PROGRAM PRG_GEM1
VAR
	{attribute 'pytmc' :=' pv: EM1L0:GEM:CNTRL:RESET;
     field: ZNAM FALSE; 
	 field: ONAM TRUE; 
	 io: io;
	'}
	bReset : BOOL; 
	{attribute 'pytmc' :=' pv: EM1L0:GEM:CNTRL:ERROR;
     field: ZNAM FALSE; 
	 field: ONAM TRUE; 
	 io: io;
	'}
	bError : BOOL; 
	{attribute 'pytmc' :=' pv: EM1L0:GEM:CNTRL:Kp1 '}
	fKp1 : REAL:= 0.5; 
	{attribute 'pytmc' :=' pv: EM1L0:GEM:CNTRL:Tn1 '}
	fTn1 : REAL:= 0.5; 
	{attribute 'pytmc' :=' pv: EM1L0:GEM:CNTRL:Kp2 '}
	fKp2 : REAL:= 0.01; 
	{attribute 'pytmc' :=' pv: EM1L0:GEM:CNTRL:Tn2 '}
	fTn2 : REAL:= 0.5; 
	arrTable_GEM1	: ARRAY[1..31,1..2] OF FLOAT;
	fManValue											: FLOAT;
	bExtrapolate										: BOOL;
	eMode							: E_CTRL_MODE;
	stCTRL_PID_PARAMS		: ST_CTRL_PID_PARAMS;
	bSync							: BOOL;
	bHold							: BOOL;
	eErrorId						: E_CTRL_ERRORCODES;
	bARWactive					: BOOL;
	(* controller *)
	fbCTRL_PID					: FB_CTRL_PID;
	bInit							: BOOL	:= TRUE;
	fbCTRL_LIN_INTERPOLATION					: FB_CTRL_LIN_INTERPOLATION;
	//stCTRL_LIN_INTERPOLATION_PARAMS		: ST_CTRL_LIN_INTERPOLATION_PARAMS;
	stCTRL_LIN_INTERPOLATION_PARAMS_GEM	: ST_CTRL_LIN_INTERPOLATION_PARAMS;
	fbCTRL_DEADBAND						: FB_CTRL_DEADBAND;
	stCTRL_DEADBAND_PARAMS			: ST_CTRL_DEADBAND_PARAMS;
		//timer to switch the pid from manual to active 5seconds??? 10 seconds???
	pid_on :TON;
	wait : time := T#10S;
FTrig: F_TRIG;	
	
	
END_VAR


(*Devices*)
(* GEM 1*)
(*Gauges*)
GEM1_GCM_41(i_rFULL_SCALE := 10.0 (*Torr*));
GEM1_GCM_42(i_rFULL_SCALE := 0.05 (*Torr*));
(*Assign reading to psuedo gauge*)
IF (GEM1_GCM_42.PG.rPRESS >0.04) THEN GEM1_GCM_40 := GEM1_GCM_42.PG;
	ELSE
	GEM1_GCM_40 := GEM1_GCM_41.PG;	
END_IF
(* N2 Cut Off Valves *)
GEM1_VVC_40(i_xExtILK_OK:= GEM1_Aperture_Closed AND GEM1_Turbo_Valves_Open AND GEM1_Turbo_Running); 

(*Flow Control Valves*)
GEM1_VCN_40 (i_xExtIlkOK := (GEM1_Aperture_Closed AND GEM1_Turbo_Valves_Open AND GEM1_Turbo_Running),// AND  GEM1_VVC_40.M_IsOpen()),
			 i_ReqPos:= fbCTRL_LIN_INTERPOLATION.fOut + fbCTRL_PID.fOut);
//GEM1_VPC_42 (i_xExtIlkOK := TRUE, i_rReqPos:= );



(*Iniitialization*)
IF bInit
THEN
	
	
	(* init array with the interpolation points  *)
	(* 	fIn					 |		fOut		*)
	arrTable_GEM1[1,1] := 0;		arrTable_GEM1[1,2] := 0;
	arrTable_GEM1[2,1] := 0.00178;		arrTable_GEM1[2,2] := 30;
	arrTable_GEM1[3,1] := 0.0025;		arrTable_GEM1[3,2] := 32;
	arrTable_GEM1[4,1] :=  0.003;	    arrTable_GEM1[4,2] := 34;
	arrTable_GEM1[5,1] :=  0.005884;	    arrTable_GEM1[5,2] := 35;
	arrTable_GEM1[6,1] := 0.0045;		arrTable_GEM1[6,2] := 42;
	arrTable_GEM1[7,1] := 0.09;		arrTable_GEM1[7,2] := 45;
	arrTable_GEM1[8,1] := 0.1;	    arrTable_GEM1[8,2] := 46;
	arrTable_GEM1[9,1] := 0.152;	    arrTable_GEM1[9,2] := 47;
	arrTable_GEM1[10,1] := 0.199;		arrTable_GEM1[10,2] := 50;
	arrTable_GEM1[11,1] := 0.24;		arrTable_GEM1[11,2] := 52;
	arrTable_GEM1[12,1] := 0.29;		arrTable_GEM1[12,2] := 54;
	arrTable_GEM1[13,1] := 0.3;		arrTable_GEM1[13,2] := 56;
	arrTable_GEM1[14,1] := 0.39;		arrTable_GEM1[14,2] := 56.5;
	arrTable_GEM1[15,1] := 0.6;		arrTable_GEM1[15,2] := 58;
	arrTable_GEM1[16,1] := 0.6929;		arrTable_GEM1[16,2] := 60;
	arrTable_GEM1[17,1] := 0.7322;		arrTable_GEM1[17,2] := 62;
	arrTable_GEM1[18,1] := 0.7928;	    arrTable_GEM1[18,2] := 64;
	arrTable_GEM1[19,1] := 0.85;;	    arrTable_GEM1[19,2] :=66;
	arrTable_GEM1[20,1] := 0.91;		arrTable_GEM1[20,2] := 68;
	arrTable_GEM1[21,1] := 1;		arrTable_GEM1[21,2] := 69;
	arrTable_GEM1[22,1] :=  1.0448;	    arrTable_GEM1[22,2] := 70;
	arrTable_GEM1[23,1] :=  1.31919;	    arrTable_GEM1[23,2] := 72;
	arrTable_GEM1[24,1] :=1.324;		arrTable_GEM1[24,2] := 73.04;
	arrTable_GEM1[25,1] :=1.71941;		arrTable_GEM1[25,2] := 73.64;
	arrTable_GEM1[26,1] := 1.81941;		arrTable_GEM1[26,2] := 74.45;
	arrTable_GEM1[27,1] :=  1.963194;		arrTable_GEM1[27,2] :=74.46;
	arrTable_GEM1[28,1] := 1.99999;	arrTable_GEM1[28,2] := 75;
	arrTable_GEM1[29,1] :=  2;		arrTable_GEM1[29,2] :=75.5;
	arrTable_GEM1[30,1] := 2.1;	arrTable_GEM1[30,2] := 75.505;
	arrTable_GEM1[31,1] := 2.2;	arrTable_GEM1[31,2] := 75.55;
	
	(* init parameter struct *)
	stCTRL_LIN_INTERPOLATION_PARAMS_GEM.tCtrlCycleTime					:= T#10ms;
	stCTRL_LIN_INTERPOLATION_PARAMS_GEM.tTaskCycleTime					:= T#10ms;
	stCTRL_LIN_INTERPOLATION_PARAMS_GEM.nDataTable_NumberOfRows		:= INT_TO_UINT(31);	


	(* init parameter struct *)
	stCTRL_PID_PARAMS.tCtrlCycleTime		:= T#10ms;
	stCTRL_PID_PARAMS.tTaskCycleTime		:= T#10ms;
	stCTRL_PID_PARAMS.fKp					:= fKp1;			(* proportional gain Kp				*)
	stCTRL_PID_PARAMS.tTn					:= T#1s;		(*  Tn									*)
	stCTRL_PID_PARAMS.tTv					:= T#200ms;	(*  Tv									*)
	stCTRL_PID_PARAMS.tTd					:= T#100ms;	(*  Td									*)
	stCTRL_PID_PARAMS.fOutMaxLimit			:=  78;			(* maximum output limit				*)
	stCTRL_PID_PARAMS.fOutMinLimit			:=  -100;			(* minimum output limit				*)

	(* set the mode to ACTIVE --> normal operation *)
	eMode							:= eCTRL_MODE_PASSIVE    ;					
	(* reset the init flag *)
	bInit							:= FALSE;
END_IF
(* set the addresses *)
stCTRL_LIN_INTERPOLATION_PARAMS_GEM.pDataTable_ADR			:= ADR(arrTable_GEM1);
stCTRL_LIN_INTERPOLATION_PARAMS_GEM.nDataTable_SIZEOF		:= SIZEOF(arrTable_GEM1);



if (GEM1_GO) THEN
	IF (bReset) THEN
		(* set the mode to RESET*)
		eMode							:= eCTRL_MODE_RESET   ;
		GEM1_VCN_40.M_ValveControl(CloseValve);
		//bReset := False;
	ELSE(* set the mode to ACTIVE --> normal operation *)
		eMode							:= eCTRL_MODE_ACTIVE   ;
		GEM1_VCN_40.M_ValveControl(PressureControl);
	END_IF
END_IF

If(FTrig.Q)THEN
		eMode							:= eCTRL_MODE_PASSIVE;
		GEM1_VCN_40.M_ValveControl(CloseValve);
		fGEM1SetpointValue :=0;
END_IF


fbCTRL_LIN_INTERPOLATION(
	fIn:= fGEM1SetpointValue , 
	fManValue:= fManValue, 
	bExtrapolate:= bExtrapolate, 
	eMode:= eMode, 
	fOut=> , 
	bInIsGreaterThanMaxElement=> , 
	bInIsLessThanMinElement=> , 
	eState=> , 
	eErrorId=> , 
	bError=> , 
	stParams:= stCTRL_LIN_INTERPOLATION_PARAMS_GEM );
	
(* Gauge selection *)
IF (fGEM1SetpointValue >0.04) THEN
	fbCTRL_PID.fActualValue := GEM1_GCM_41.PG.rPRESS;
ELSE
	fbCTRL_PID.fActualValue := GEM1_GCM_42.PG.rPRESS;
END_IF

	
(* call controller *)
fbCTRL_PID(		fSetpointValue		:= fGEM1SetpointValue,
					fActualValue		:= ,
					fManSyncValue	:= ,
					bSync				:= bSync,
					eMode				:= eMode,
					bHold				:= bHold,
					stParams			:= stCTRL_PID_PARAMS,
					fOut				=>  ,
					bARWactive		=> bARWactive,
					eErrorId			=> eErrorId,
					bError				=> 
				);


	
(*deadband/clipper *)

(* call function block *)
stCTRL_DEADBAND_PARAMS.fThreshold	:=  fGEM1SetpointValue*0.01 ;
(*fbCTRL_DEADBAND	(	fIn					:= ,
					stParams			:= stCTRL_DEADBAND_PARAMS,
					bInIsUnderThreshold => ,
					eErrorId			=> ,
					bError				=> 
				);*)
				
bError := fbCTRL_PID.bError OR fbCTRL_LIN_INTERPOLATION.bError;


// or NOT???

//stCTRL_PID_PARAMS.bDInTheFeedbackPath := fbCTRL_DEADBAND.bInIsUnderThreshold;


//timer
//pid_on(IN:=, PT:= wait, Q=>, ET =>);
//IF (pid_on.Q) THEN eMode:= eCTRL_MODE_ACTIVE; pid_on.IN := FALSE; END_IF; //eCTRL_MODE_TUNE????

FTRIG(CLK := GEM1_GO);

END_PROGRAM

(* stored: Version 1.1.0.1, ProductVersion 3.1.4022.18
   POU PRG_GEM1: Id {b5aed3c6-13be-428f-86ce-8bd830676022}, SpecialFunc None *)
